TYPE ST_ServiceStatusBase :
STRUCT
	Busy : BOOL;
	Done : BOOL;
	Error : BOOL;
	Aborted : BOOL;
	ErrorId : UDINT;
	State : E_PackMLState;
END_STRUCT
END_TYPE

(* stored: Version 1.1.0.1, ProductVersion 3.1.4026.18
   DUT ST_ServiceStatusBase: Id {696bda33-0a33-48b0-8ccd-362e4a358520} *)
